# EPICS alarm handler configuration: mps_database/bare/alarms/areas/mpln_dog_mp02.alhConfig
GROUP NULL MPLN:DOG:MP02:1
$ALIAS MPS Link Node 73
$GUIDANCE
LTUH MPS
   Group Name: MPLN:DOG:MP02:1
   Summary PV:  MPLN:DOG:MP02:1:STATSUMY
$END
CHANNEL  MPLN:DOG:MP02:1    MPLN:DOG:MP02:1:MPS_EN_RBV		-----
CHANNEL  MPLN:DOG:MP02:1    MPLN:DOG:MP02:1:LC1_MODE_RBV		-----
